FUNCTION_BLOCK FB_MotionLogger IMPLEMENTS I_MotionLogger
VAR_INPUT
END_VAR
VAR_OUTPUT
END_VAR
VAR
END_VAR

END_FUNCTION_BLOCK

(* stored: Version 1.1.0.1
   POU FB_MotionLogger: Id {b6dde3c0-50f4-4c2e-b05e-f0f55b5fa75d}, SpecialFunc None *)
